FUNCTION_BLOCK AirPiston IMPLEMENTS I_ContinuousDrive
VAR_INPUT
	bEnable : BOOL;
END_VAR
VAR_OUTPUT
	valveExtend AT %Q* : BOOL;
	valveRetract AT %Q* : BOOL;
END_VAR
VAR
	mode : (HOLD, IN, OUT);
	brakePulse : TP; //generates the retraction pulse
END_VAR
VAR_STAT CONSTANT
	brakeWidth : TIME := T#650MS;
END_VAR

IF NOT bEnable THEN
	stop();
	RETURN;
END_IF

brakePulse(IN:= , PT:= brakeWidth, Q=> , ET=> ); //reversal to act as brake
brakePulse.IN := brakePulse.IN AND brakePulse.Q; //automatically turn off pulse

override();

CASE mode OF
	HOLD:
		valveExtend := FALSE;
		valveRetract := FALSE;
		
	IN:
		valveExtend := TRUE;
		valveRetract := FALSE;
		
	OUT:
		valveExtend := FALSE;
		valveRetract := TRUE;
		
END_CASE

valveRetract := valveRetract OR brakePulse.Q; //from mode or brake

PROPERTY Active : BOOL
GET
Active :=
	mode <> HOLD AND
	valveExtend OR valveRetract;
END_GET
END_PROPERTY

PROPERTY Error : BOOL
GET
END_GET
END_PROPERTY

METHOD extend : BOOL
VAR_INPUT
END_VAR
mode := IN;
END_METHOD

{attribute 'TcRpcEnable'}
METHOD moveContinuous : BOOL
VAR_INPUT
	newDirection : MC_Direction;
END_VAR
IF newDirection = MC_Positive_Direction THEN
	retract();
ELSIF newDirection = MC_Negative_Direction THEN
	extend();
END_IF
END_METHOD

METHOD PROTECTED override : BOOL
VAR_INPUT
END_VAR
(*
IF brakePulse.Q THEN
	mode := HOLD;
END_IF

IF AtHome AND (valveRetract OR mode = OUT) THEN
	mode := HOLD;
	
ELSIF AtInnerLimit AND (valveExtend OR mode = IN) THEN	
	brakePulse.IN := useBrake;
	mode := HOLD;
END_IF


IF NOT bEnable THEN
	stop();
END_IF
*)

IF Error THEN
	stop();
	reset();
END_IF
END_METHOD

METHOD reset : BOOL
VAR_INPUT
END_VAR
stop();
END_METHOD

METHOD retract : BOOL
VAR_INPUT
END_VAR
mode := OUT;
END_METHOD

METHOD stop : BOOL
VAR_INPUT
END_VAR
valveExtend := FALSE;
valveRetract := FALSE;
mode := HOLD;

stop := TRUE;
END_METHOD

METHOD toHome : BOOL
VAR_INPUT
END_VAR
mode := OUT;
END_METHOD

END_FUNCTION_BLOCK

(* stored: Version 1.1.0.1, ProductVersion 3.1.4024.11
   POU AirPiston: Id {b09c4aa7-1ed0-4b4c-a588-8d696c2002d5}, SpecialFunc None
   Folder Hidden: Id {52fbe06a-8565-410c-8614-2f4bf25bac46}
   Folder Properties: Id {0b37a229-5e45-4012-856f-0994150a2a37}
   Property Active: Id {e0c19726-96c6-4b23-9713-d5fa5c51978b}
   Get Get: Id {3ffc0014-b13e-48a4-a011-a47bf2912abc}
   Property Error: Id {4b3c428e-5925-4b68-abda-e333fd39ea6c}
   Get Get: Id {426bfa48-a9b6-45da-b528-8a66be7702b3}
   Method extend: Id {8e9fb730-3c54-4958-b095-df03386fa45e}
   Method moveContinuous: Id {b1d0f050-e29a-41a5-a0da-5771c5954de0}
   Method override: Id {b5d71d3e-17bd-4818-8115-1f45d76b4b10}
   Method reset: Id {49e8bda4-f9c4-4a67-8236-4f3ea27ddf4a}
   Method retract: Id {f3abddeb-a229-4f56-aaa9-218f8f27dc5d}
   Method stop: Id {65d9d8a8-5400-4c12-8076-ebbf37d71867}
   Method toHome: Id {97e8c420-493b-4b68-859a-2d794017b851} *)
